Staubli VAL3: SetFrame.dtx

mdesc mNomSpeed
public pointRx pFrameRefPt[3]
  [0] = {fatherId=world[0]}
  [1] = {fatherId=world[0]}
  [2] = {fatherId=world[0]}
tool tTool = {fatherId=flange[0], ioLink=valve1}
num nFrame1Err
string sOffSet[6]
trsf trOffset
frame fFrame1 = {fatherId=world[0]}
string sThreeOffset[3]
bool bSame
string sCutPosStatus
string sEmptyOrNotC[3]
string sItem[6]
num nItem[6]
num nSelectedPt
num nMin[6]
num nMax[6]
public bool bFrameSave
bool bExit
num nWorkingMode
num nStatus
frame fFrameRef = {fatherId=world[0]}
trsf trOffSetOut
num nDia
bool bOk
pointRx pPointCenter = {fatherId=world[0]}
string sButton[2]
bool bFrameTeach
